(* CODESYS project tank1.project

Project tree, tasks and I/O mapping:
  Device : CODESYS Control Win V3, 3S - Smart Software Solutions GmbH, version 3.5.3.50
    application Application
      libraries: Standard, 3.5.2.0 (System)
      task MainTask (cyclic, interval t#20ms, priority 1) calls Levels, Main, Simulate
      program Levels [FBD]
      program Main [SFC]: Init_level
      function block Process [SFC]
      global variables GVL
      program Simulate [ST]
  libraries: VisuSymbols, 3.5.10.0 (System)
  visualisation Visualization
  text list GlobalTextList
*)

// Device/Application/GVL
VAR_GLOBAL
	run: BOOL;
	level: REAL;
	empty: BOOL;
	full: BOOL;
	in_valve: BOOL;
	out_valve: BOOL;
	resistor: BOOL;
	temperature: REAL;
	hot: BOOL;
END_VAR

VAR_GLOBAL
	step: INT;
END_VAR

// Device/Application/Levels
PROGRAM Levels
VAR
END_VAR

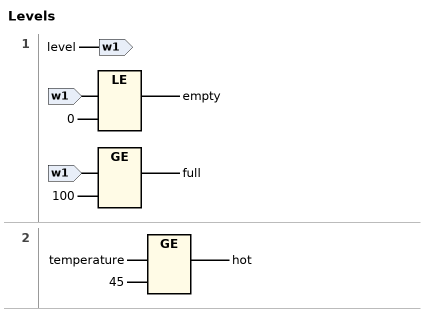
// NETWORK 1
empty := level <= 0;
full := level >= 100;

// NETWORK 2
hot := temperature >= 45;

END_PROGRAM

// Device/Application/Main
PROGRAM Main
VAR
	process: Process;
END_VAR

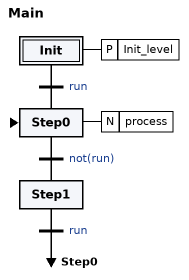
INITIAL_STEP Init:
    Init_level(P);
END_STEP
TRANSITION FROM Init TO Step0
    := run;
END_TRANSITION
STEP Step0:
    process(N);
END_STEP
TRANSITION FROM Step0 TO Step1
    := not(run);
END_TRANSITION
STEP Step1:
END_STEP
TRANSITION FROM Step1 TO Step0
    := run;
END_TRANSITION

ACTION Init_level:
level := 0;
END_ACTION

END_PROGRAM

// Device/Application/Process
FUNCTION_BLOCK Process

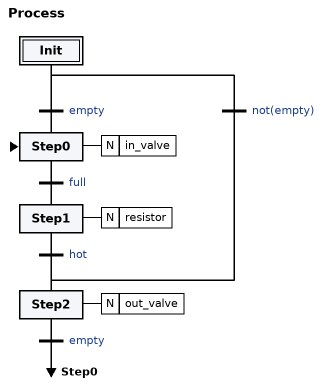
INITIAL_STEP Init:
END_STEP
TRANSITION FROM Init TO Step0
    := empty;
END_TRANSITION
STEP Step0:
    in_valve(N);
END_STEP
TRANSITION FROM Step0 TO Step1
    := full;
END_TRANSITION
STEP Step1:
    resistor(N);
END_STEP
TRANSITION FROM Step1 TO Step2
    := hot;
END_TRANSITION
TRANSITION FROM Init TO Step2
    := not(empty);
END_TRANSITION
STEP Step2:
    out_valve(N);
END_STEP
TRANSITION FROM Step2 TO Step0
    := empty;
END_TRANSITION

END_FUNCTION_BLOCK

// Device/Application/Simulate
PROGRAM Simulate
VAR
END_VAR

(* simulates level increase or decrease *)
(* according to valve status *)
IF (in_valve) THEN
   level := level + 0.2;
END_IF;
IF (out_valve) THEN
	IF level >= 0.2 THEN
   		level := level - 0.2;
	ELSE
		level := 0;
	END_IF
END_IF;

(* simulate temperature increase *)
(* according to resistor status *)
IF (resistor) THEN
	temperature := temperature + 0.1;
END_IF
IF (empty) THEN
	temperature := 21;
END_IF

END_PROGRAM

// /Visualization
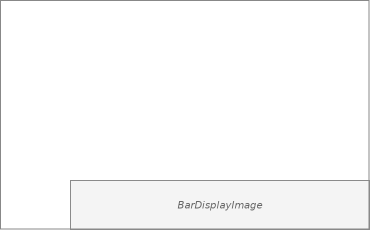
VISUALIZATION Visualization  // 370x230
    BarDisplayImage (70,180 300x50), value: temperature, style: BarDisplayImage-Gray, scale format: %.1f, scale 0..100
END_VISUALIZATION
